// LS Electric XG5000 project: 과년69_3(수정)
// PLC NewPLC
// module base 0 slot 0: 입출력 모듈:XBC-DR20S (DC 24V 입력 12점, 릴레이 출력 8점)

PROGRAM NewProgram (task: 스캔 프로그램)

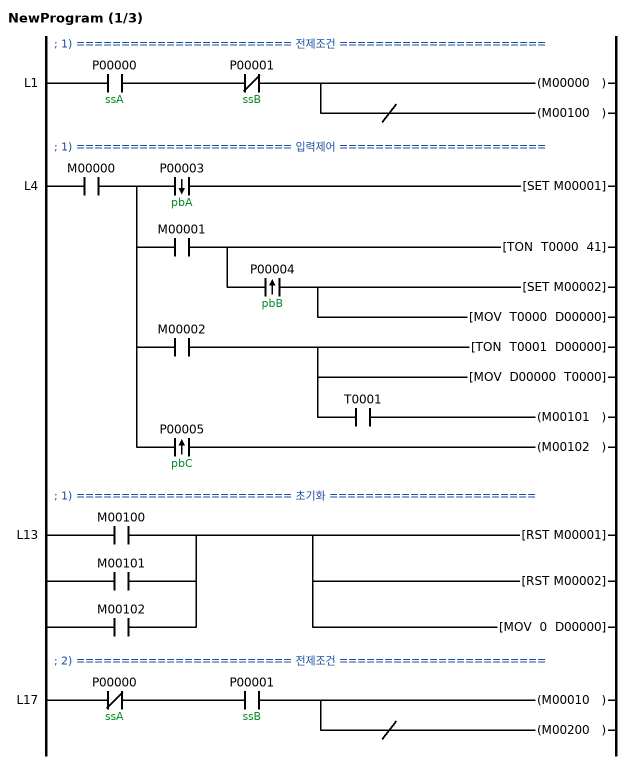
// 1) ======================== 전제조건 =======================
; L1
LOAD      P00000	// ssA
AND NOT   P00001	// ssB
OUT       M00000
NOT
OUT       M00100
// 1) ======================== 입력제어 =======================
; L4
LOAD      M00000
MPUSH
ANDN      P00003	// pbA
SET       M00001
MLOAD
AND       M00001
TON       T0000 41
ANDP      P00004	// pbB
SET       M00002
MOV       T0000 D00000
MLOAD
AND       M00002
TON       T0001 D00000
MOV       D00000 T0000
AND       T0001
OUT       M00101
MPOP
ANDP      P00005	// pbC
OUT       M00102
// 1) ======================== 초기화 =======================
; L13
LOAD      M00100
OR        M00101
OR        M00102
RST       M00001
RST       M00002
MOV       0 D00000
// 2) ======================== 전제조건 =======================
; L17
LOAD NOT  P00000	// ssA
AND       P00001	// ssB
OUT       M00010
NOT
OUT       M00200

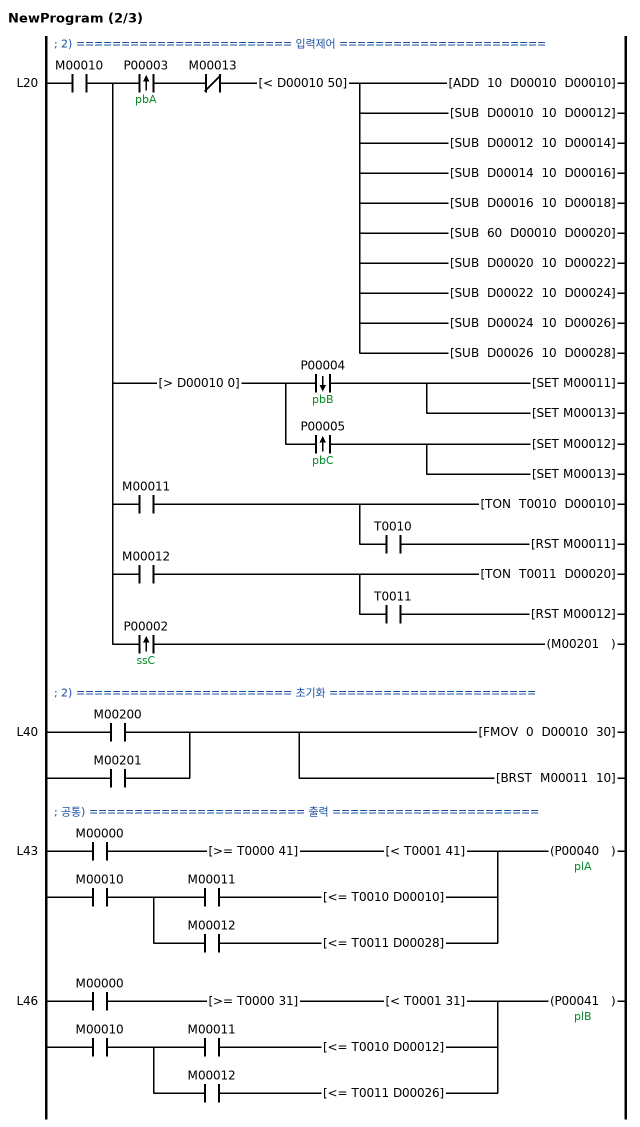
// 2) ======================== 입력제어 =======================
; L20
LOAD      M00010
MPUSH
ANDP      P00003	// pbA
AND NOT   M00013
AND<      D00010 50
ADD       10 D00010 D00010
SUB       D00010 10 D00012
SUB       D00012 10 D00014
SUB       D00014 10 D00016
SUB       D00016 10 D00018
SUB       60 D00010 D00020
SUB       D00020 10 D00022
SUB       D00022 10 D00024
SUB       D00024 10 D00026
SUB       D00026 10 D00028
MLOAD
AND>      D00010 0
MPUSH
ANDN      P00004	// pbB
SET       M00011
SET       M00013
MPOP
ANDP      P00005	// pbC
SET       M00012
SET       M00013
MLOAD
AND       M00011
TON       T0010 D00010
AND       T0010
RST       M00011
MLOAD
AND       M00012
TON       T0011 D00020
AND       T0011
RST       M00012
MPOP
ANDP      P00002	// ssC
OUT       M00201
// 2) ======================== 초기화 =======================
; L40
LOAD      M00200
OR        M00201
FMOV      0 D00010 30
BRST      M00011 10
// 공통) ======================== 출력 =======================
; L43
LOAD      M00000
AND>=     T0000 41
AND<      T0001 41
LOAD      M00010
LOAD      M00011
AND<=     T0010 D00010
LOAD      M00012
AND<=     T0011 D00028
OR LOAD
AND LOAD
OR LOAD
OUT       P00040	// plA
; L46
LOAD      M00000
AND>=     T0000 31
AND<      T0001 31
LOAD      M00010
LOAD      M00011
AND<=     T0010 D00012
LOAD      M00012
AND<=     T0011 D00026
OR LOAD
AND LOAD
OR LOAD
OUT       P00041	// plB

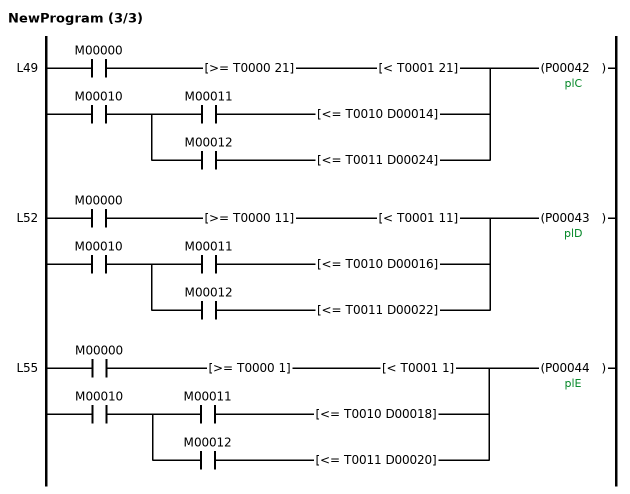
; L49
LOAD      M00000
AND>=     T0000 21
AND<      T0001 21
LOAD      M00010
LOAD      M00011
AND<=     T0010 D00014
LOAD      M00012
AND<=     T0011 D00024
OR LOAD
AND LOAD
OR LOAD
OUT       P00042	// plC
; L52
LOAD      M00000
AND>=     T0000 11
AND<      T0001 11
LOAD      M00010
LOAD      M00011
AND<=     T0010 D00016
LOAD      M00012
AND<=     T0011 D00022
OR LOAD
AND LOAD
OR LOAD
OUT       P00043	// plD
; L55
LOAD      M00000
AND>=     T0000 1
AND<      T0001 1
LOAD      M00010
LOAD      M00011
AND<=     T0010 D00018
LOAD      M00012
AND<=     T0011 D00020
OR LOAD
AND LOAD
OR LOAD
OUT       P00044	// plE